FUNCTION_BLOCK FB_State EXTENDS FB_Object IMPLEMENTS I_State
VAR
    _bQueryRes:             BOOL;
END_VAR

METHOD OnEntry
VAR_INPUT
END_VAR
END_METHOD

METHOD OnExit
VAR_INPUT
END_VAR
END_METHOD

END_FUNCTION_BLOCK

(* stored: Version 1.1.0.1, ProductVersion 3.1.4024.12
   POU FB_State: Id {78f523dd-b10e-48af-9696-be0082d49d72}, SpecialFunc None
   Method OnEntry: Id {4827bf9d-4efc-4534-b327-d8caa3685450}
   Method OnExit: Id {75371a96-da45-4aac-8255-1aa82ef7ac67} *)
